(* PLC project Communication Blocks, OpenPLC Communication Blocks Library 1.0, author Thiago Alves *)
(* stored: creationDateTime 2022-11-11T02:33:11, modificationDateTime 2022-11-11T02:33:11 *)

(* Connect to a remote TCP server when CONNECT is TRUE. Upon success, this block returns the connection ID on SOCKET_ID. If SOCKET_ID is less than zero, then the connection was not successfull *)
FUNCTION_BLOCK TCP_CONNECT
  VAR_INPUT
    CONNECT : BOOL;
    IP_ADDRESS : STRING;
    PORT : INT;
  END_VAR
  VAR_OUTPUT
    SOCKET_ID : INT;
  END_VAR

            SOCKET_ID := 0;
          
END_FUNCTION_BLOCK

(* Send a message to a remote device using TCP/IP when SEND is TRUE. SOCKET_ID must receive a connection ID from a successfull connection using the TCP_Connect block. BYTES_SENT returns the number of bytes sent to the remote device. If BYTES_SENT is less than zero then an error occurred while trying to send the message *)
FUNCTION_BLOCK TCP_SEND
  VAR_INPUT
    SEND : BOOL;
    SOCKET_ID : INT;
    MSG : STRING;
  END_VAR
  VAR_OUTPUT
    BYTES_SENT : INT;
  END_VAR

            BYTES_SENT := 0;
          
END_FUNCTION_BLOCK

(* Send a message to a remote device using TCP/IP when SEND is TRUE. SOCKET_ID must receive a connection ID from a successfull connection using the TCP_Connect block. BYTES_RECEIVED returns the number of bytes received from the remote device. MSG is a String containing the message received *)
FUNCTION_BLOCK TCP_RECEIVE
  VAR_INPUT
    RECEIVE : BOOL;
    SOCKET_ID : INT;
  END_VAR
  VAR_OUTPUT
    BYTES_RECEIVED : INT;
    MSG : STRING;
  END_VAR

            BYTES_RECEIVED := 0;
          
END_FUNCTION_BLOCK

(* Close the TCP connection with the remote server. If SUCCESS is less than zero, then the connection was not successfully closed, or the connection does not exist anymore. *)
FUNCTION_BLOCK TCP_CLOSE
  VAR_INPUT
    CLOSE : BOOL;
    SOCKET_ID : INT;
  END_VAR
  VAR_OUTPUT
    SUCCESS : INT;
  END_VAR

            SUCCESS := 0;
          
END_FUNCTION_BLOCK
